// TIA Portal V16 export
// export: Created 2025-05-30T16:36:20.2354944Z, ExportSetting WithDefaults, DisplayName Totally Integrated Automation Portal, DisplayVersion V16, DisplayName TIA Portal Version Control Interface, DisplayVersion V16, DisplayName TIA Portal Openness, DisplayVersion V16, DisplayName STEP 7 Professional, DisplayVersion V16, DisplayName STEP 7 Safety, DisplayVersion V16, DisplayName WinCC Advanced, DisplayVersion V16
DATA_BLOCK "Alarms"   // DB24
VERSION : 0.1
// stored: AutoNumber true, IsOnlyStoredInLoadMemory false, IsWriteProtectedInAS false
   VAR
      AlarmStruct : Struct
         Alarm_Product_Not_Position : Bool;
         Alarm_Axis_Not_Position : Bool;
         Alarm_Drive1 : Bool;
         Alarm_Drive2 : Bool;
         Alarm_Drive3 : Bool;
         Alarm_Drive4 : Bool;
         Alarm_Drive5 : Bool;
         "Alarm_To_Many_Products_Reset_Counter!" : Bool;
      END_STRUCT;
      AlarmsWord : Word;
      HMI_Alarm_Drive1 : Word;
      HMI_Alarm_Drive2 : Word;
      HMI_Alarm_Drive3 : Word;
      HMI_Alarm_Drive4 : Word;
      HMI_Alarm_Drive5 : Word;
   END_VAR
BEGIN
END_DATA_BLOCK
